KUKA KRL data list: BrakeTestSelfTest.dat

&ACCESS RVO
DEFDAT BrakeTestSelfTest PUBLIC

INT simulateBrakeVel    = 100
INT simulateBrakeTorque = 50
INT simulateBrakeIndex  = 2

ENDDAT
